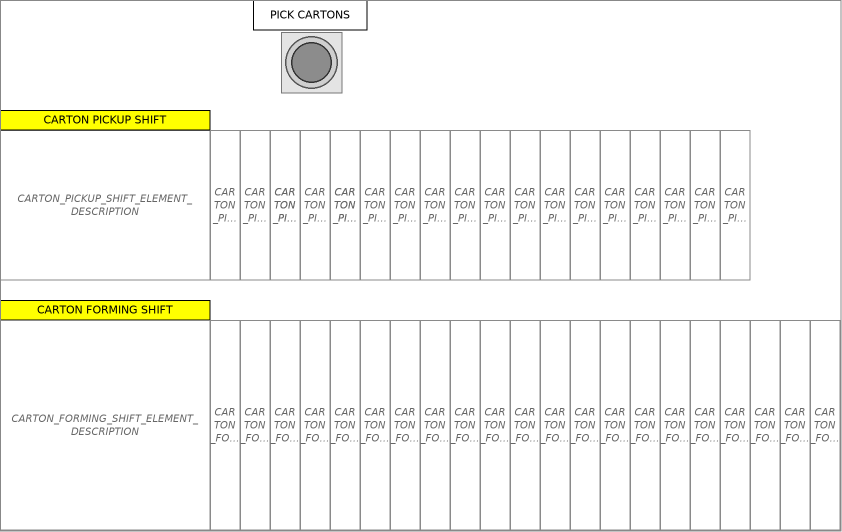
VISUALIZATION CARTON_SHIFT  // 842x532
    Frame (0,130 210x150)
        shows CARTON_PICKUP_SHIFT_ELEMENT_DESCRIPTION()
    Rectangle (0,110 210x20), "CARTON PICKUP SHIFT"
    Frame (210,130 30x150)
        shows CARTON_PICKUP_SHIFT_ELEMENT(index := 95)
    Frame (240,130 30x150)
        shows CARTON_PICKUP_SHIFT_ELEMENT(index := 96)
    Frame (270,130 30x150)
        shows CARTON_PICKUP_SHIFT_ELEMENT(index := 1)
    Frame (270,130 30x150)
        shows CARTON_PICKUP_SHIFT_ELEMENT(index := 97)
    Frame (300,130 30x150)
        shows CARTON_PICKUP_SHIFT_ELEMENT(index := 98)
    Frame (330,130 30x150)
        shows CARTON_PICKUP_SHIFT_ELEMENT(index := 1)
    Frame (330,130 30x150)
        shows CARTON_PICKUP_SHIFT_ELEMENT(index := 99)
    Frame (360,130 30x150)
        shows CARTON_PICKUP_SHIFT_ELEMENT(index := 100)
    Frame (390,130 30x150)
        shows CARTON_PICKUP_SHIFT_ELEMENT(index := 101)
    Frame (420,130 30x150)
        shows CARTON_PICKUP_SHIFT_ELEMENT(index := 102)
    Frame (450,130 30x150)
        shows CARTON_PICKUP_SHIFT_ELEMENT(index := 103)
    Frame (480,130 30x150)
        shows CARTON_PICKUP_SHIFT_ELEMENT(index := 104)
    Frame (510,130 30x150)
        shows CARTON_PICKUP_SHIFT_ELEMENT(index := 105)
    Frame (540,130 30x150)
        shows CARTON_PICKUP_SHIFT_ELEMENT(index := 106)
    Frame (570,130 30x150)
        shows CARTON_PICKUP_SHIFT_ELEMENT(index := 107)
    Frame (600,130 30x150)
        shows CARTON_PICKUP_SHIFT_ELEMENT(index := 108)
    Frame (630,130 30x150)
        shows CARTON_PICKUP_SHIFT_ELEMENT(index := 109)
    Frame (660,130 30x150)
        shows CARTON_PICKUP_SHIFT_ELEMENT(index := 110)
    Frame (690,130 30x150)
        shows CARTON_PICKUP_SHIFT_ELEMENT(index := 111)
    Frame (720,130 30x150)
        shows CARTON_PICKUP_SHIFT_ELEMENT(index := 112)
    Rectangle (0,300 210x20), "CARTON FORMING SHIFT"
    Frame (0,320 210x210)
        shows CARTON_FORMING_SHIFT_ELEMENT_DESCRIPTION()
    Frame (210,320 30x210)
        shows CARTON_FORMING_SHIFT_ELEMENT(index := 100)
    Frame (240,320 30x210)
        shows CARTON_FORMING_SHIFT_ELEMENT(index := 101)
    Frame (270,320 30x210)
        shows CARTON_FORMING_SHIFT_ELEMENT(index := 102)
    Frame (300,320 30x210)
        shows CARTON_FORMING_SHIFT_ELEMENT(index := 103)
    Frame (330,320 30x210)
        shows CARTON_FORMING_SHIFT_ELEMENT(index := 104)
    Frame (360,320 30x210)
        shows CARTON_FORMING_SHIFT_ELEMENT(index := 105)
    Frame (390,320 30x210)
        shows CARTON_FORMING_SHIFT_ELEMENT(index := 106)
    Frame (420,320 30x210)
        shows CARTON_FORMING_SHIFT_ELEMENT(index := 107)
    Frame (450,320 30x210)
        shows CARTON_FORMING_SHIFT_ELEMENT(index := 108)
    Frame (480,320 30x210)
        shows CARTON_FORMING_SHIFT_ELEMENT(index := 109)
    Frame (510,320 30x210)
        shows CARTON_FORMING_SHIFT_ELEMENT(index := 110)
    Frame (540,320 30x210)
        shows CARTON_FORMING_SHIFT_ELEMENT(index := 111)
    Frame (570,320 30x210)
        shows CARTON_FORMING_SHIFT_ELEMENT(index := 112)
    Frame (600,320 30x210)
        shows CARTON_FORMING_SHIFT_ELEMENT(index := 113)
    Frame (630,320 30x210)
        shows CARTON_FORMING_SHIFT_ELEMENT(index := 114)
    Frame (660,320 30x210)
        shows CARTON_FORMING_SHIFT_ELEMENT(index := 115)
    Frame (690,320 30x210)
        shows CARTON_FORMING_SHIFT_ELEMENT(index := 116)
    Frame (720,320 30x210)
        shows CARTON_FORMING_SHIFT_ELEMENT(index := 117)
    PushSwitch (279,32 65x61), variable: wu_cartonPickup_drums_suction.debug, behaviour: TOGGLE, style: Switch-PushSwitch-Gray
    Rectangle (253,0 114x30), "PICK CARTONS"
    Frame (750,320 30x210)
        shows CARTON_FORMING_SHIFT_ELEMENT(index := 118)
    Frame (780,320 30x210)
        shows CARTON_FORMING_SHIFT_ELEMENT(index := 119)
    Frame (810,320 30x210)
        shows CARTON_FORMING_SHIFT_ELEMENT(index := 120)
END_VISUALIZATION

(* stored: Version 1.1.0.1, ProductVersion 3.1.4024.3
   Visu CARTON_SHIFT: Id {e2cacecf-9db3-4d43-891d-9f006d86697a} *)
